// TIA Portal V17 export
// export: Created 2024-09-02T12:50:00.3255564Z, ExportSetting WithDefaults, DisplayName Totally Integrated Automation Portal, DisplayVersion V17, DisplayName TIA Portal Openness, DisplayVersion V17, DisplayName TIA Portal Version Control Interface, DisplayVersion V17, DisplayName STEP 7 Professional, DisplayVersion V17, DisplayName STEP 7 Safety, DisplayVersion V17, DisplayName WinCC Professional, DisplayVersion V17
FUNCTION_BLOCK "GraFB_Hand_31_40"   // FB1173, GRAPH
TITLE = GRAPH FB
AUTHOR : OlegFuehrus
FAMILY : SK
NAME : SK
VERSION : 0.1
// Hand functions / Handfunktionen
// stored: AcknowledgeErrorsRequired true, AutoNumber true, ExtensionBlockName LTLL_ManualGraphExt, GraphVersion 4.0, InitialValuesAcquisition false, IsIECCheckEnabled false, LanguageInNetworks LAD, LockOperatingMode false, PermanentILProcessingInMANMode true, SetENOAutomatically false, SkipSteps false, UDAEnableTagReadback false, WithAlarmHandling true
   // inherited from GRAPH_BASE
   VAR
      OFF_SQ_BASE : Bool;
   END_VAR
   VAR_INPUT
      OFF_SQ : Bool;
      INIT_SQ : Bool;
      ACK_EF : Bool;
      S_PREV : Bool;
      S_NEXT : Bool;
      SW_AUTO : Bool;
      SW_TAP : Bool;
      SW_MAN : Bool;
      S_SEL : Int;
      S_ON : Bool;
      S_OFF : Bool;
      T_PUSH : Bool;
   END_VAR
   VAR_OUTPUT
      S_NO : Int;
      S_MORE : Bool;
      S_ACTIVE : Bool;
      ERR_FLT : Bool;
      AUTO_ON : Bool;
      TAP_ON : Bool;
      MAN_ON : Bool;
   END_VAR
   VAR
      extBlock { S7_SetPoint := 'True'} : "LTLL_ManualGraphExt";
   END_VAR
   VAR_TEMP
      t_FrgHand : Bool;   // Freigabe Handbetrieb / Enable manual operation
      t_Service : Bool;   // Servicebetrieb aktiv / Service operation active
   END_VAR
BEGIN
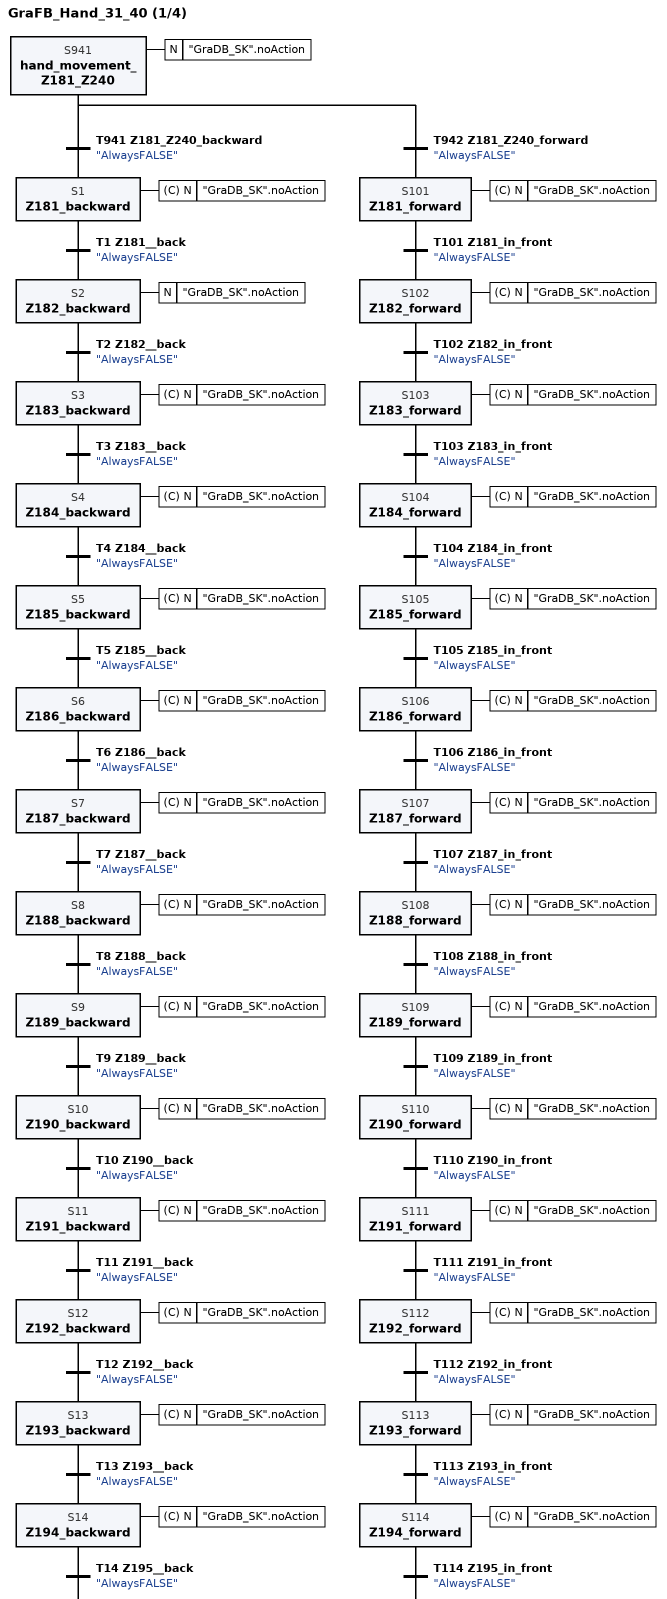
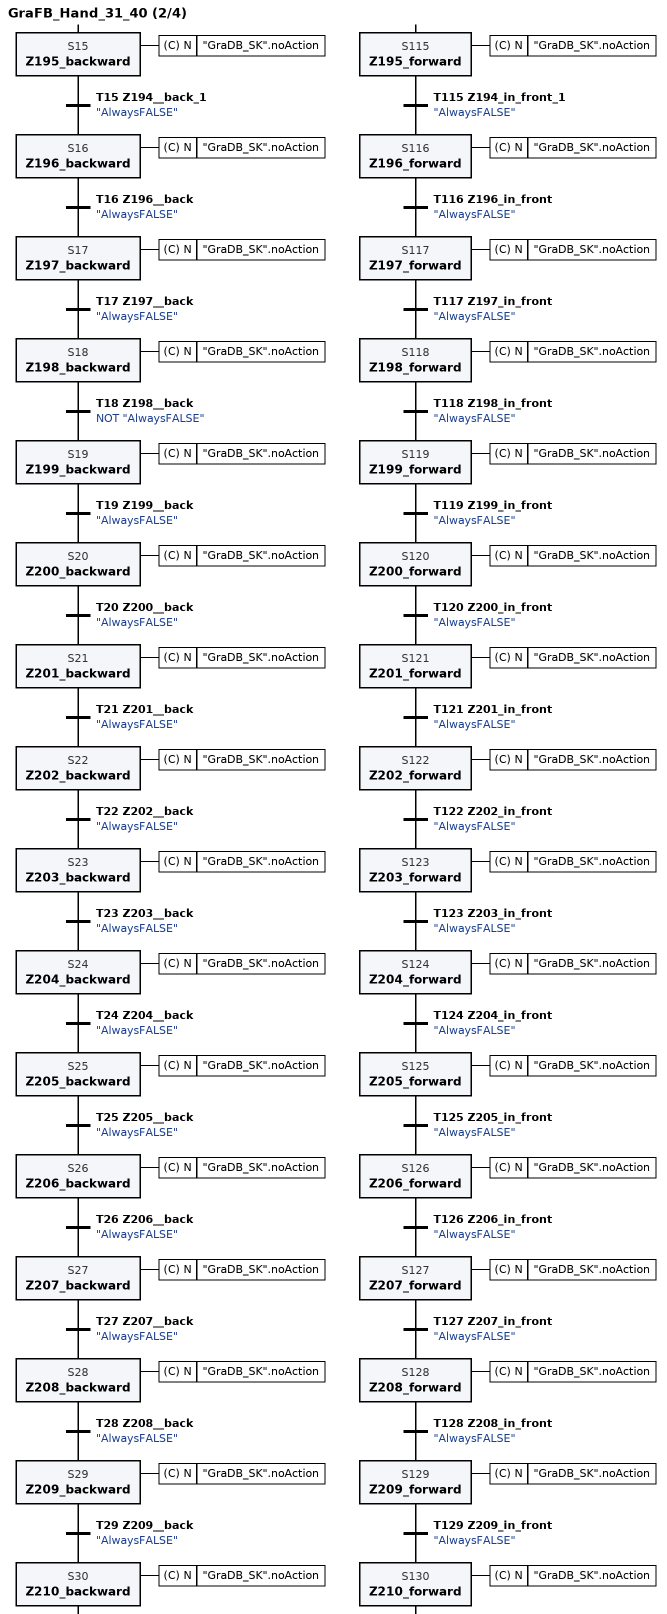
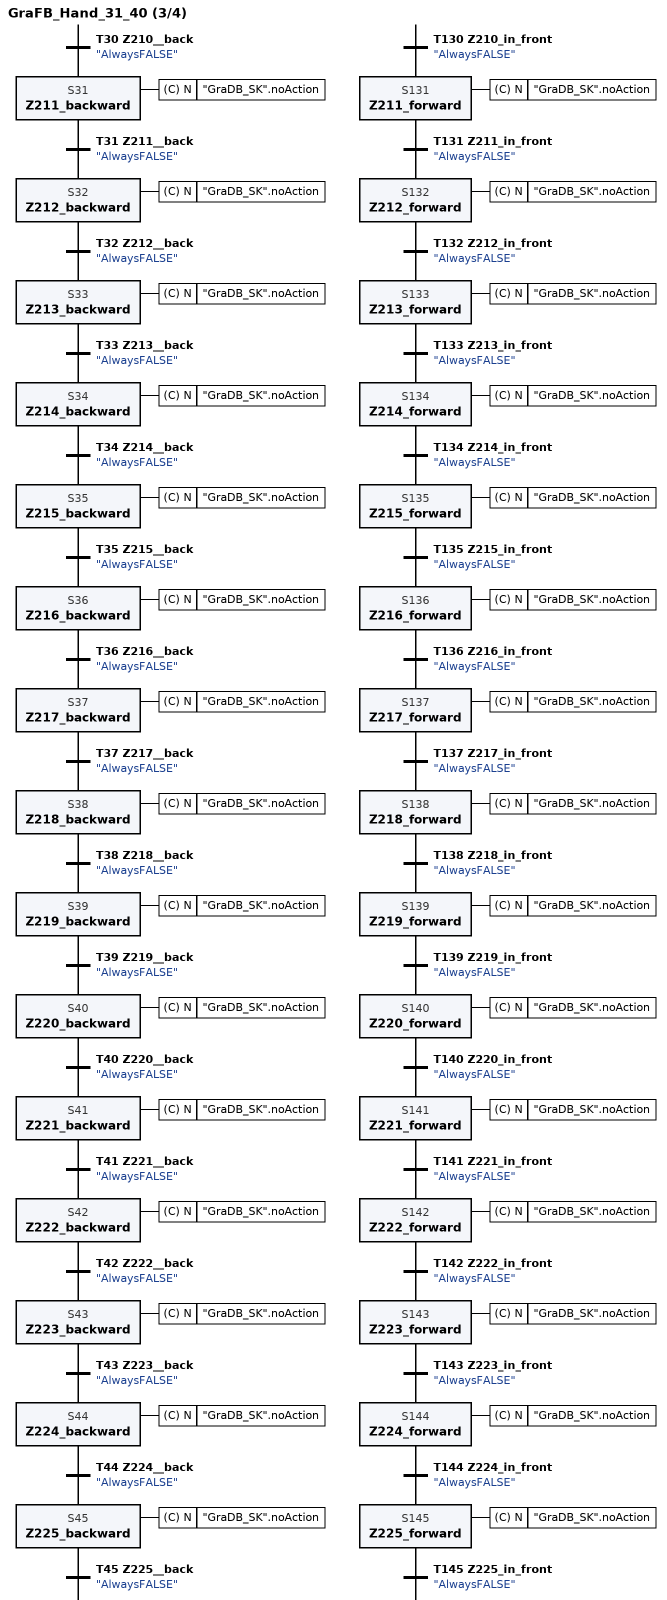
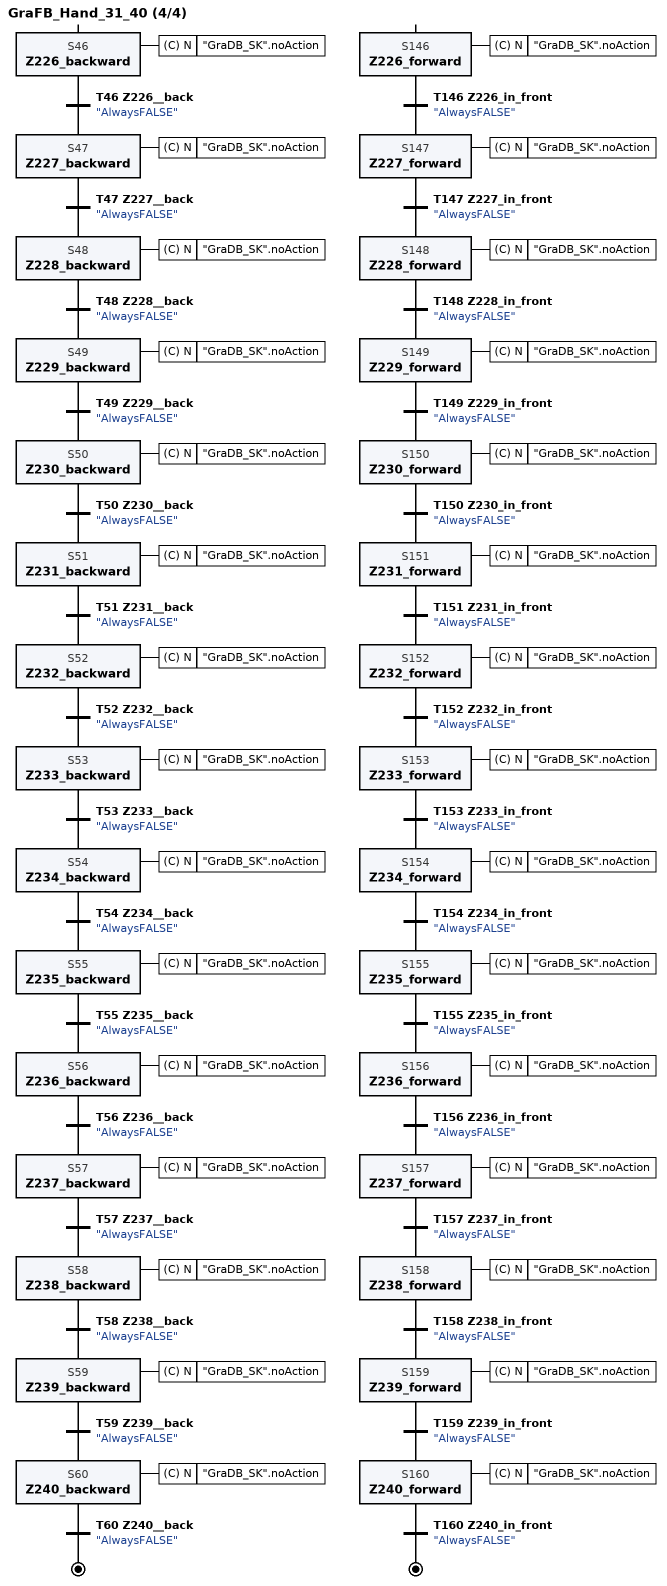
   // permanent pre-instructions
   NETWORK 1
   TITLE = HMI Lite Pass on data / HMI Lite Daten weiterreichen
      #extBlock.input := "LTLL_ManualGraphControl_OP70".screen[0].input;
   NETWORK 2
   TITLE = Instance DB Name query and pass on / Instanz DB Name abfragen und weiterreichen
      GetInstanceName(size := 0, OUT => #extBlock.input.instanceName);
   NETWORK 3
   TITLE = Interlocks Permanent machining, manual Approve and service / Interlocks Permanent Bearbeiten, Handfreigabe und Service
      IF NOT #RT_DATA.MOP.IL_PERM THEN #RT_DATA.MOP.IL_PERM := TRUE; END_IF;
      #t_FrgHand := "AnwDB_OperatingModes_OP70".BA[0]."mode_hand+start";
      #t_Service := "AnwDB_OperatingModes_OP70".BA[0].mode_service;

   // sequencer 1: Sequencer 1
   STEP hand_movement_Z181_Z240:   // S941, max time T#10S, warning time T#7S: Step commentary / Schrittkommentar
      interlock C := (none);   // hand_bereich_Z001_Z005
      supervision V := (none);   // hand_bereich_Z001_Z005
              N    "GraDB_SK".noAction
   END_STEP
   TRANSITION Z181_Z240_backward FROM hand_movement_Z181_Z240 TO Z181_backward   // T941
      := "AlwaysFALSE";
   END_TRANSITION
   TRANSITION Z181_Z240_forward FROM hand_movement_Z181_Z240 TO Z181_forward   // T942
      := "AlwaysFALSE";
   END_TRANSITION
   STEP Z181_backward:   // S1, max time T#10S, warning time T#7S
      interlock C := "AlwaysFALSE";   // Z181_zur
      supervision V := NOT #Z181__back.TT AND (#Z181_backward.T > T#5S);   // Z181_zur
      (C)     N    "GraDB_SK".noAction
   END_STEP
   TRANSITION Z181__back FROM Z181_backward TO Z182_backward   // T1
      := "AlwaysFALSE";
   END_TRANSITION
   STEP Z182_backward:   // S2, max time T#10S, warning time T#7S
      interlock C := "AlwaysFALSE";   // Z182_zur
      supervision V := NOT #Z182__back.TT AND (#Z182_backward.T > T#5S);   // Z182_zur
              N    "GraDB_SK".noAction
   END_STEP
   TRANSITION Z182__back FROM Z182_backward TO Z183_backward   // T2
      := "AlwaysFALSE";
   END_TRANSITION
   STEP Z183_backward:   // S3, max time T#10S, warning time T#7S
      interlock C := "AlwaysFALSE";   // Z183_zur
      supervision V := NOT #Z183__back.TT AND (#Z183_backward.T > T#5S);   // Z183_zur
      (C)     N    "GraDB_SK".noAction
   END_STEP
   TRANSITION Z183__back FROM Z183_backward TO Z184_backward   // T3
      := "AlwaysFALSE";
   END_TRANSITION
   STEP Z184_backward:   // S4, max time T#10S, warning time T#7S
      interlock C := "AlwaysFALSE";   // Z184_zur
      supervision V := NOT #Z184__back.TT AND (#Z184_backward.T > T#5S);   // Z184_zur
      (C)     N    "GraDB_SK".noAction
   END_STEP
   TRANSITION Z184__back FROM Z184_backward TO Z185_backward   // T4
      := "AlwaysFALSE";
   END_TRANSITION
   STEP Z185_backward:   // S5, max time T#10S, warning time T#7S
      interlock C := "AlwaysFALSE";   // Z185_zur
      supervision V := NOT #Z185__back.TT AND (#Z185_backward.T > T#5S);   // Z185_zur
      (C)     N    "GraDB_SK".noAction
   END_STEP
   TRANSITION Z185__back FROM Z185_backward TO Z186_backward   // T5
      := "AlwaysFALSE";
   END_TRANSITION
   STEP Z181_forward:   // S101, max time T#10S, warning time T#7S
      interlock C := "AlwaysFALSE";   // Z181_vor
      supervision V := NOT #Z181_in_front.TT AND (#Z181_forward.T > T#5S);   // Z181_vor
      (C)     N    "GraDB_SK".noAction
   END_STEP
   TRANSITION Z181_in_front FROM Z181_forward TO Z182_forward   // T101
      := "AlwaysFALSE";
   END_TRANSITION
   STEP Z182_forward:   // S102, max time T#10S, warning time T#7S
      interlock C := "AlwaysFALSE";   // Z182_vor
      supervision V := NOT #Z182_in_front.TT AND (#Z182_forward.T > T#5S);   // Z182_vor
      (C)     N    "GraDB_SK".noAction
   END_STEP
   TRANSITION Z182_in_front FROM Z182_forward TO Z183_forward   // T102
      := "AlwaysFALSE";
   END_TRANSITION
   STEP Z183_forward:   // S103, max time T#10S, warning time T#7S
      interlock C := "AlwaysFALSE";   // Z183_vor
      supervision V := NOT #Z183_in_front.TT AND (#Z183_forward.T > T#5S);   // Z183_vor
      (C)     N    "GraDB_SK".noAction
   END_STEP
   TRANSITION Z183_in_front FROM Z183_forward TO Z184_forward   // T103
      := "AlwaysFALSE";
   END_TRANSITION
   STEP Z184_forward:   // S104, max time T#10S, warning time T#7S
      interlock C := "AlwaysFALSE";   // Z184_vor
      supervision V := NOT #Z184_in_front.TT AND (#Z184_forward.T > T#5S);   // Z184_vor
      (C)     N    "GraDB_SK".noAction
   END_STEP
   TRANSITION Z184_in_front FROM Z184_forward TO Z185_forward   // T104
      := "AlwaysFALSE";
   END_TRANSITION
   STEP Z185_forward:   // S105, max time T#10S, warning time T#7S
      interlock C := "AlwaysFALSE";   // Z185_vor
      supervision V := NOT #Z185_in_front.TT AND (#Z185_forward.T > T#20S);   // Z185_vor
      (C)     N    "GraDB_SK".noAction
   END_STEP
   TRANSITION Z185_in_front FROM Z185_forward TO Z186_forward   // T105
      := "AlwaysFALSE";
   END_TRANSITION
   STEP Z186_backward:   // S6, max time T#10S, warning time T#7S: Cross transport 2 / Quertransport 2
      interlock C := "AlwaysFALSE";   // Z186_zur
      supervision V := NOT #Z186__back.TT AND (#Z186_backward.T > T#5S);   // Z186_zur
      (C)     N    "GraDB_SK".noAction
   END_STEP
   TRANSITION Z186__back FROM Z186_backward TO Z187_backward   // T6
      := "AlwaysFALSE";
   END_TRANSITION
   STEP Z187_backward:   // S7, max time T#10S, warning time T#7S
      interlock C := "AlwaysFALSE";   // Z187_zur
      supervision V := NOT #Z187__back.TT AND (#Z187_backward.T > T#5S);   // Z187_zur
      (C)     N    "GraDB_SK".noAction
   END_STEP
   TRANSITION Z187__back FROM Z187_backward TO Z188_backward   // T7
      := "AlwaysFALSE";
   END_TRANSITION
   STEP Z188_backward:   // S8, max time T#10S, warning time T#7S
      interlock C := "AlwaysFALSE";   // Z188_zur
      supervision V := NOT #Z188__back.TT AND (#Z188_backward.T > T#5S);   // Z188_zur
      (C)     N    "GraDB_SK".noAction
   END_STEP
   TRANSITION Z188__back FROM Z188_backward TO Z189_backward   // T8
      := "AlwaysFALSE";
   END_TRANSITION
   STEP Z189_backward:   // S9, max time T#10S, warning time T#7S
      interlock C := "AlwaysFALSE";   // Z189_zur
      supervision V := NOT #Z189__back.TT AND (#Z189_backward.T > T#5S);   // Z189_zur
      (C)     N    "GraDB_SK".noAction
   END_STEP
   TRANSITION Z189__back FROM Z189_backward TO Z190_backward   // T9
      := "AlwaysFALSE";
   END_TRANSITION
   STEP Z190_backward:   // S10, max time T#10S, warning time T#7S
      interlock C := "AlwaysFALSE";   // Z190_zur
      supervision V := NOT #Z190__back.TT AND (#Z190_backward.T > T#5S);   // Z190_zur
      (C)     N    "GraDB_SK".noAction
   END_STEP
   TRANSITION Z190__back FROM Z190_backward TO Z191_backward   // T10
      := "AlwaysFALSE";
   END_TRANSITION
   STEP Z186_forward:   // S106, max time T#10S, warning time T#7S
      interlock C := "AlwaysFALSE";   // Z186_vor
      supervision V := NOT #Z186_in_front.TT AND (#Z186_forward.T > T#5S);   // Z186_vor
      (C)     N    "GraDB_SK".noAction
   END_STEP
   TRANSITION Z186_in_front FROM Z186_forward TO Z187_forward   // T106
      := "AlwaysFALSE";
   END_TRANSITION
   STEP Z187_forward:   // S107, max time T#10S, warning time T#7S
      interlock C := "AlwaysFALSE";   // Z187_vor
      supervision V := NOT #Z187_in_front.TT AND (#Z187_forward.T > T#5S);   // Z187_vor
      (C)     N    "GraDB_SK".noAction
   END_STEP
   TRANSITION Z187_in_front FROM Z187_forward TO Z188_forward   // T107
      := "AlwaysFALSE";
   END_TRANSITION
   STEP Z188_forward:   // S108, max time T#10S, warning time T#7S
      interlock C := "AlwaysFALSE";   // Z188_vor
      supervision V := NOT #Z188_in_front.TT AND (#Z188_forward.T > T#5S);   // Z188_vor
      (C)     N    "GraDB_SK".noAction
   END_STEP
   TRANSITION Z188_in_front FROM Z188_forward TO Z189_forward   // T108
      := "AlwaysFALSE";
   END_TRANSITION
   STEP Z189_forward:   // S109, max time T#10S, warning time T#7S
      interlock C := "AlwaysFALSE";   // Z189_vor
      supervision V := NOT #Z189_in_front.TT AND (#Z189_forward.T > T#5S);   // Z189_vor
      (C)     N    "GraDB_SK".noAction
   END_STEP
   TRANSITION Z189_in_front FROM Z189_forward TO Z190_forward   // T109
      := "AlwaysFALSE";
   END_TRANSITION
   STEP Z190_forward:   // S110, max time T#10S, warning time T#7S
      interlock C := "AlwaysFALSE";   // Z190_vor
      supervision V := NOT #Z190_in_front.TT AND (#Z190_forward.T > T#5S);   // Z190_vor
      (C)     N    "GraDB_SK".noAction
   END_STEP
   TRANSITION Z190_in_front FROM Z190_forward TO Z191_forward   // T110
      := "AlwaysFALSE";
   END_TRANSITION
   STEP Z191_backward:   // S11, max time T#10S, warning time T#7S
      interlock C := "AlwaysFALSE";   // Z191_zur
      supervision V := NOT #Z191__back.TT AND (#Z191_backward.T > T#5S);   // Z191_zur
      (C)     N    "GraDB_SK".noAction
   END_STEP
   TRANSITION Z191__back FROM Z191_backward TO Z192_backward   // T11
      := "AlwaysFALSE";
   END_TRANSITION
   STEP Z192_backward:   // S12, max time T#10S, warning time T#7S
      interlock C := "AlwaysFALSE";   // Z192_zur
      supervision V := NOT #Z192__back.TT AND (#Z192_backward.T > T#5S);   // Z192_zur
      (C)     N    "GraDB_SK".noAction
   END_STEP
   TRANSITION Z192__back FROM Z192_backward TO Z193_backward   // T12
      := "AlwaysFALSE";
   END_TRANSITION
   STEP Z193_backward:   // S13, max time T#10S, warning time T#7S
      interlock C := "AlwaysFALSE";   // Z193_zur
      supervision V := NOT #Z193__back.TT AND (#Z193_backward.T > T#5S);   // Z193_zur
      (C)     N    "GraDB_SK".noAction
   END_STEP
   TRANSITION Z193__back FROM Z193_backward TO Z194_backward   // T13
      := "AlwaysFALSE";
   END_TRANSITION
   STEP Z194_backward:   // S14, max time T#10S, warning time T#7S
      interlock C := "AlwaysFALSE";   // Z194_zur
      supervision V := NOT #Z195__back.TT AND (#Z194_backward.T > T#5S);   // Z194_zur
      (C)     N    "GraDB_SK".noAction
   END_STEP
   TRANSITION Z195__back FROM Z194_backward TO Z195_backward   // T14
      := "AlwaysFALSE";
   END_TRANSITION
   STEP Z195_backward:   // S15, max time T#10S, warning time T#7S
      interlock C := "AlwaysFALSE";   // Z195_zur
      supervision V := NOT #Z196__back.TT AND (#Z195_backward.T > T#5S);   // Z195_zur
      (C)     N    "GraDB_SK".noAction
   END_STEP
   TRANSITION Z194__back_1 FROM Z195_backward TO Z196_backward   // T15
      := "AlwaysFALSE";
   END_TRANSITION
   STEP Z191_forward:   // S111, max time T#10S, warning time T#7S
      interlock C := "AlwaysFALSE";   // Z191_vor
      supervision V := NOT #Z191_in_front.TT AND (#Z191_forward.T > T#5S);   // Z191_vor
      (C)     N    "GraDB_SK".noAction
   END_STEP
   TRANSITION Z191_in_front FROM Z191_forward TO Z192_forward   // T111
      := "AlwaysFALSE";
   END_TRANSITION
   STEP Z192_forward:   // S112, max time T#10S, warning time T#7S
      interlock C := "AlwaysFALSE";   // Z192_vor
      supervision V := NOT #Z192_in_front.TT AND (#Z192_forward.T > T#5S);   // Z192_vor
      (C)     N    "GraDB_SK".noAction
   END_STEP
   TRANSITION Z192_in_front FROM Z192_forward TO Z193_forward   // T112
      := "AlwaysFALSE";
   END_TRANSITION
   STEP Z193_forward:   // S113, max time T#10S, warning time T#7S
      interlock C := "AlwaysFALSE";   // Z193_vor
      supervision V := NOT #Z193_in_front.TT AND (#Z193_forward.T > T#5S);   // Z193_vor
      (C)     N    "GraDB_SK".noAction
   END_STEP
   TRANSITION Z193_in_front FROM Z193_forward TO Z194_forward   // T113
      := "AlwaysFALSE";
   END_TRANSITION
   STEP Z194_forward:   // S114, max time T#10S, warning time T#7S
      interlock C := "AlwaysFALSE";   // Z194_vor
      supervision V := NOT #Z195_in_front.TT AND (#Z194_forward.T > T#5S);   // Z194_vor
      (C)     N    "GraDB_SK".noAction
   END_STEP
   TRANSITION Z195_in_front FROM Z194_forward TO Z195_forward   // T114
      := "AlwaysFALSE";
   END_TRANSITION
   STEP Z195_forward:   // S115, max time T#10S, warning time T#7S
      interlock C := "AlwaysFALSE";   // Z195_vor
      supervision V := NOT #Z196_in_front.TT AND (#Z195_forward.T > T#5S);   // Z195_vor
      (C)     N    "GraDB_SK".noAction
   END_STEP
   TRANSITION Z194_in_front_1 FROM Z195_forward TO Z196_forward   // T115
      := "AlwaysFALSE";
   END_TRANSITION
   STEP Z196_backward:   // S16, max time T#10S, warning time T#7S
      interlock C := "AlwaysFALSE";   // Z196_zur
      supervision V := NOT #Z196__back.TT AND (#Z196_backward.T > T#5S);   // Z196_zur
      (C)     N    "GraDB_SK".noAction
   END_STEP
   TRANSITION Z196__back FROM Z196_backward TO Z197_backward   // T16
      := "AlwaysFALSE";
   END_TRANSITION
   STEP Z197_backward:   // S17, max time T#10S, warning time T#7S
      interlock C := "AlwaysFALSE";   // Z197_zur
      supervision V := NOT #Z197__back.TT AND (#Z197_backward.T > T#5S);   // Z197_zur
      (C)     N    "GraDB_SK".noAction
   END_STEP
   TRANSITION Z197__back FROM Z197_backward TO Z198_backward   // T17
      := "AlwaysFALSE";
   END_TRANSITION
   STEP Z198_backward:   // S18, max time T#10S, warning time T#7S
      interlock C := "AlwaysFALSE";   // Z198_zur
      supervision V := NOT #Z198__back.TT AND (#Z198_backward.T > T#5S);   // Z198_zur
      (C)     N    "GraDB_SK".noAction
   END_STEP
   TRANSITION Z198__back FROM Z198_backward TO Z199_backward   // T18
      := NOT "AlwaysFALSE";
   END_TRANSITION
   STEP Z199_backward:   // S19, max time T#10S, warning time T#7S
      interlock C := "AlwaysFALSE";   // Z199_zur
      supervision V := NOT #Z199__back.TT AND (#Z199_backward.T > T#5S);   // Z199_zur
      (C)     N    "GraDB_SK".noAction
   END_STEP
   TRANSITION Z199__back FROM Z199_backward TO Z200_backward   // T19
      := "AlwaysFALSE";
   END_TRANSITION
   STEP Z200_backward:   // S20, max time T#10S, warning time T#7S
      interlock C := "AlwaysFALSE";   // Z200_zur
      supervision V := NOT #Z200__back.TT AND (#Z200_backward.T > T#5S);   // Z2000_zur
      (C)     N    "GraDB_SK".noAction
   END_STEP
   TRANSITION Z200__back FROM Z200_backward TO Z201_backward   // T20
      := "AlwaysFALSE";
   END_TRANSITION
   STEP Z196_forward:   // S116, max time T#10S, warning time T#7S
      interlock C := "AlwaysFALSE";   // Z196_vor
      supervision V := NOT #Z196_in_front.TT AND (#Z196_forward.T > T#5S);   // Z196_vor
      (C)     N    "GraDB_SK".noAction
   END_STEP
   TRANSITION Z196_in_front FROM Z196_forward TO Z197_forward   // T116
      := "AlwaysFALSE";
   END_TRANSITION
   STEP Z197_forward:   // S117, max time T#10S, warning time T#7S
      interlock C := "AlwaysFALSE";   // Z197_vor
      supervision V := NOT #Z197_in_front.TT AND (#Z197_forward.T > T#5S);   // Z197_vor
      (C)     N    "GraDB_SK".noAction
   END_STEP
   TRANSITION Z197_in_front FROM Z197_forward TO Z198_forward   // T117
      := "AlwaysFALSE";
   END_TRANSITION
   STEP Z198_forward:   // S118, max time T#10S, warning time T#7S
      interlock C := "AlwaysFALSE";   // Z198_vor
      supervision V := NOT #Z198_in_front.TT AND (#Z198_forward.T > T#5S);   // Z198_vor
      (C)     N    "GraDB_SK".noAction
   END_STEP
   TRANSITION Z198_in_front FROM Z198_forward TO Z199_forward   // T118
      := "AlwaysFALSE";
   END_TRANSITION
   STEP Z199_forward:   // S119, max time T#10S, warning time T#7S
      interlock C := "AlwaysFALSE";   // Z199_vor
      supervision V := NOT #Z199_in_front.TT AND (#Z199_forward.T > T#5S);   // Z199_vor
      (C)     N    "GraDB_SK".noAction
   END_STEP
   TRANSITION Z199_in_front FROM Z199_forward TO Z200_forward   // T119
      := "AlwaysFALSE";
   END_TRANSITION
   STEP Z200_forward:   // S120, max time T#10S, warning time T#7S
      interlock C := "AlwaysFALSE";   // Z200_vor
      supervision V := NOT #Z200_in_front.TT AND (#Z200_forward.T > T#5S);   // Z200_vor
      (C)     N    "GraDB_SK".noAction
   END_STEP
   TRANSITION Z200_in_front FROM Z200_forward TO Z201_forward   // T120
      := "AlwaysFALSE";
   END_TRANSITION
   STEP Z201_backward:   // S21, max time T#10S, warning time T#7S
      interlock C := "AlwaysFALSE";   // Z201_zur
      supervision V := NOT #Z201__back.TT AND (#Z201_backward.T > T#10S);   // Z201_zur
      (C)     N    "GraDB_SK".noAction
   END_STEP
   TRANSITION Z201__back FROM Z201_backward TO Z202_backward   // T21
      := "AlwaysFALSE";
   END_TRANSITION
   STEP Z202_backward:   // S22, max time T#10S, warning time T#7S
      interlock C := "AlwaysFALSE";   // Z202_zur
      supervision V := NOT #Z202__back.TT AND (#Z202_backward.T > T#10S);   // Z202_zur
      (C)     N    "GraDB_SK".noAction
   END_STEP
   TRANSITION Z202__back FROM Z202_backward TO Z203_backward   // T22
      := "AlwaysFALSE";
   END_TRANSITION
   STEP Z203_backward:   // S23, max time T#10S, warning time T#7S
      interlock C := "AlwaysFALSE";   // Z203_zur
      supervision V := NOT #Z203__back.TT AND (#Z203_backward.T > T#10S);   // Z203_zur
      (C)     N    "GraDB_SK".noAction
   END_STEP
   TRANSITION Z203__back FROM Z203_backward TO Z204_backward   // T23
      := "AlwaysFALSE";
   END_TRANSITION
   STEP Z204_backward:   // S24, max time T#10S, warning time T#7S
      interlock C := "AlwaysFALSE";   // Z204_zur
      supervision V := NOT #Z204__back.TT AND (#Z204_backward.T > T#5S);   // Z204_zur
      (C)     N    "GraDB_SK".noAction
   END_STEP
   TRANSITION Z204__back FROM Z204_backward TO Z205_backward   // T24
      := "AlwaysFALSE";
   END_TRANSITION
   STEP Z205_backward:   // S25, max time T#10S, warning time T#7S
      interlock C := "AlwaysFALSE";   // Z205_zur
      supervision V := NOT #Z205__back.TT AND (#Z205_backward.T > T#5S);   // Z205_zur
      (C)     N    "GraDB_SK".noAction
   END_STEP
   TRANSITION Z205__back FROM Z205_backward TO Z206_backward   // T25
      := "AlwaysFALSE";
   END_TRANSITION
   STEP Z201_forward:   // S121, max time T#10S, warning time T#7S
      interlock C := "AlwaysFALSE";   // Z201_vor
      supervision V := NOT #Z201_in_front.TT AND (#Z201_forward.T > T#5S);   // Z201_vor
      (C)     N    "GraDB_SK".noAction
   END_STEP
   TRANSITION Z201_in_front FROM Z201_forward TO Z202_forward   // T121
      := "AlwaysFALSE";
   END_TRANSITION
   STEP Z202_forward:   // S122, max time T#10S, warning time T#7S
      interlock C := "AlwaysFALSE";   // Z202_vor
      supervision V := NOT #Z202_in_front.TT AND (#Z202_forward.T > T#10S);   // Z202_vor
      (C)     N    "GraDB_SK".noAction
   END_STEP
   TRANSITION Z202_in_front FROM Z202_forward TO Z203_forward   // T122
      := "AlwaysFALSE";
   END_TRANSITION
   STEP Z203_forward:   // S123, max time T#10S, warning time T#7S
      interlock C := "AlwaysFALSE";   // Z203_vor
      supervision V := NOT #Z203_in_front.TT AND (#Z203_forward.T > T#10S);   // Z203_vor
      (C)     N    "GraDB_SK".noAction
   END_STEP
   TRANSITION Z203_in_front FROM Z203_forward TO Z204_forward   // T123
      := "AlwaysFALSE";
   END_TRANSITION
   STEP Z204_forward:   // S124, max time T#10S, warning time T#7S
      interlock C := "AlwaysFALSE";   // Z204_vor
      supervision V := NOT #Z204_in_front.TT AND (#Z204_forward.T > T#5S);   // Z204_vor
      (C)     N    "GraDB_SK".noAction
   END_STEP
   TRANSITION Z204_in_front FROM Z204_forward TO Z205_forward   // T124
      := "AlwaysFALSE";
   END_TRANSITION
   STEP Z205_forward:   // S125, max time T#10S, warning time T#7S
      interlock C := "AlwaysFALSE";   // Z205_vor
      supervision V := NOT #Z205_in_front.TT AND (#Z205_forward.T > T#5S);   // Z205_vor
      (C)     N    "GraDB_SK".noAction
   END_STEP
   TRANSITION Z205_in_front FROM Z205_forward TO Z206_forward   // T125
      := "AlwaysFALSE";
   END_TRANSITION
   STEP Z206_backward:   // S26, max time T#10S, warning time T#7S
      interlock C := "AlwaysFALSE";   // Z206_zur
      supervision V := NOT #Z206__back.TT AND (#Z206_backward.T > T#5S);   // Z206_zur
      (C)     N    "GraDB_SK".noAction
   END_STEP
   TRANSITION Z206__back FROM Z206_backward TO Z207_backward   // T26
      := "AlwaysFALSE";
   END_TRANSITION
   STEP Z207_backward:   // S27, max time T#10S, warning time T#7S
      interlock C := "AlwaysFALSE";   // Z207_zur
      supervision V := NOT #Z207__back.TT AND (#Z207_backward.T > T#5S);   // Z207_zur
      (C)     N    "GraDB_SK".noAction
   END_STEP
   TRANSITION Z207__back FROM Z207_backward TO Z208_backward   // T27
      := "AlwaysFALSE";
   END_TRANSITION
   STEP Z208_backward:   // S28, max time T#10S, warning time T#7S
      interlock C := "AlwaysFALSE";   // Z208_zur
      supervision V := NOT #Z208__back.TT AND (#Z208_backward.T > T#5S);   // Z208_zur
      (C)     N    "GraDB_SK".noAction
   END_STEP
   TRANSITION Z208__back FROM Z208_backward TO Z209_backward   // T28
      := "AlwaysFALSE";
   END_TRANSITION
   STEP Z209_backward:   // S29, max time T#10S, warning time T#7S
      interlock C := "AlwaysFALSE";   // Z209_zur
      supervision V := NOT #Z209__back.TT AND (#Z209_backward.T > T#5S);   // Z209_zur
      (C)     N    "GraDB_SK".noAction
   END_STEP
   TRANSITION Z209__back FROM Z209_backward TO Z210_backward   // T29
      := "AlwaysFALSE";
   END_TRANSITION
   STEP Z210_backward:   // S30, max time T#10S, warning time T#7S
      interlock C := "AlwaysFALSE";   // Z210_zur
      supervision V := NOT #Z210__back.TT AND (#Z210_backward.T > T#5S);   // Z210_zur
      (C)     N    "GraDB_SK".noAction
   END_STEP
   TRANSITION Z210__back FROM Z210_backward TO Z211_backward   // T30
      := "AlwaysFALSE";
   END_TRANSITION
   STEP Z206_forward:   // S126, max time T#10S, warning time T#7S
      interlock C := "AlwaysFALSE";   // Z206_vor
      supervision V := NOT #Z206_in_front.TT AND (#Z206_forward.T > T#5S);   // Z206_vor
      (C)     N    "GraDB_SK".noAction
   END_STEP
   TRANSITION Z206_in_front FROM Z206_forward TO Z207_forward   // T126
      := "AlwaysFALSE";
   END_TRANSITION
   STEP Z207_forward:   // S127, max time T#10S, warning time T#7S
      interlock C := "AlwaysFALSE";   // Z207_vor
      supervision V := NOT #Z207_in_front.TT AND (#Z207_forward.T > T#5S);   // Z207_vor
      (C)     N    "GraDB_SK".noAction
   END_STEP
   TRANSITION Z207_in_front FROM Z207_forward TO Z208_forward   // T127
      := "AlwaysFALSE";
   END_TRANSITION
   STEP Z208_forward:   // S128, max time T#10S, warning time T#7S
      interlock C := "AlwaysFALSE";   // Z208_vor
      supervision V := NOT #Z208_in_front.TT AND (#Z208_forward.T > T#5S);   // Z208_vor
      (C)     N    "GraDB_SK".noAction
   END_STEP
   TRANSITION Z208_in_front FROM Z208_forward TO Z209_forward   // T128
      := "AlwaysFALSE";
   END_TRANSITION
   STEP Z209_forward:   // S129, max time T#10S, warning time T#7S
      interlock C := "AlwaysFALSE";   // Z209_vor
      supervision V := NOT #Z209_in_front.TT AND (#Z209_forward.T > T#5S);   // Z209_vor
      (C)     N    "GraDB_SK".noAction
   END_STEP
   TRANSITION Z209_in_front FROM Z209_forward TO Z210_forward   // T129
      := "AlwaysFALSE";
   END_TRANSITION
   STEP Z210_forward:   // S130, max time T#10S, warning time T#7S
      interlock C := "AlwaysFALSE";   // Z210_vor
      supervision V := NOT #Z210_in_front.TT AND (#Z210_forward.T > T#5S);   // Z210_vor
      (C)     N    "GraDB_SK".noAction
   END_STEP
   TRANSITION Z210_in_front FROM Z210_forward TO Z211_forward   // T130
      := "AlwaysFALSE";
   END_TRANSITION
   STEP Z211_backward:   // S31, max time T#10S, warning time T#7S: Step commentary / Schrittkommentar
      interlock C := "AlwaysFALSE";   // Z211_zur
      supervision V := NOT #Z211__back.TT AND (#Z211_backward.T > T#5S);   // Z211_zur
      (C)     N    "GraDB_SK".noAction
   END_STEP
   TRANSITION Z211__back FROM Z211_backward TO Z212_backward   // T31
      := "AlwaysFALSE";
   END_TRANSITION
   STEP Z212_backward:   // S32, max time T#10S, warning time T#7S: Step commentary / Schrittkommentar
      interlock C := "AlwaysFALSE";   // Z212_zur
      supervision V := NOT #Z212__back.TT AND (#Z212_backward.T > T#5S);   // Z212_zur
      (C)     N    "GraDB_SK".noAction
   END_STEP
   TRANSITION Z212__back FROM Z212_backward TO Z213_backward   // T32
      := "AlwaysFALSE";
   END_TRANSITION
   STEP Z213_backward:   // S33, max time T#10S, warning time T#7S: Step commentary / Schrittkommentar
      interlock C := "AlwaysFALSE";   // Z213_zur
      supervision V := NOT #Z213__back.TT AND (#Z213_backward.T > T#5S);   // Z213_zur
      (C)     N    "GraDB_SK".noAction
   END_STEP
   TRANSITION Z213__back FROM Z213_backward TO Z214_backward   // T33
      := "AlwaysFALSE";
   END_TRANSITION
   STEP Z214_backward:   // S34, max time T#10S, warning time T#7S: Step commentary / Schrittkommentar
      interlock C := "AlwaysFALSE";   // Z034_zur
      supervision V := NOT #Z214__back.TT AND (#Z214_backward.T > T#5S);   // Z034_zur
      (C)     N    "GraDB_SK".noAction
   END_STEP
   TRANSITION Z214__back FROM Z214_backward TO Z215_backward   // T34
      := "AlwaysFALSE";
   END_TRANSITION
   STEP Z215_backward:   // S35, max time T#10S, warning time T#7S: Step commentary / Schrittkommentar
      interlock C := "AlwaysFALSE";   // Z215_zur
      supervision V := NOT #Z215__back.TT AND (#Z215_backward.T > T#5S);   // Z215_zur
      (C)     N    "GraDB_SK".noAction
   END_STEP
   TRANSITION Z215__back FROM Z215_backward TO Z216_backward   // T35
      := "AlwaysFALSE";
   END_TRANSITION
   STEP Z211_forward:   // S131, max time T#10S, warning time T#7S: Step commentary / Schrittkommentar
      interlock C := "AlwaysFALSE";   // Z211_vor
      supervision V := NOT #Z211_in_front.TT AND (#Z211_forward.T > T#5S);   // Z211_vor
      (C)     N    "GraDB_SK".noAction
   END_STEP
   TRANSITION Z211_in_front FROM Z211_forward TO Z212_forward   // T131
      := "AlwaysFALSE";
   END_TRANSITION
   STEP Z212_forward:   // S132, max time T#10S, warning time T#7S: Step commentary / Schrittkommentar
      interlock C := "AlwaysFALSE";   // Z212_vor
      supervision V := NOT #Z212_in_front.TT AND (#Z212_forward.T > T#5S);   // Z212_vor
      (C)     N    "GraDB_SK".noAction
   END_STEP
   TRANSITION Z212_in_front FROM Z212_forward TO Z213_forward   // T132
      := "AlwaysFALSE";
   END_TRANSITION
   STEP Z213_forward:   // S133, max time T#10S, warning time T#7S: Step commentary / Schrittkommentar
      interlock C := "AlwaysFALSE";   // Z213_vor
      supervision V := NOT #Z213_in_front.TT AND (#Z213_forward.T > T#5S);   // Z213_vor
      (C)     N    "GraDB_SK".noAction
   END_STEP
   TRANSITION Z213_in_front FROM Z213_forward TO Z214_forward   // T133
      := "AlwaysFALSE";
   END_TRANSITION
   STEP Z214_forward:   // S134, max time T#10S, warning time T#7S: Step commentary / Schrittkommentar
      interlock C := "AlwaysFALSE";   // Z034_vor
      supervision V := NOT #Z214_in_front.TT AND (#Z214_forward.T > T#5S);   // Z034_vor
      (C)     N    "GraDB_SK".noAction
   END_STEP
   TRANSITION Z214_in_front FROM Z214_forward TO Z215_forward   // T134
      := "AlwaysFALSE";
   END_TRANSITION
   STEP Z215_forward:   // S135, max time T#10S, warning time T#7S: Step commentary / Schrittkommentar
      interlock C := "AlwaysFALSE";   // Z215_vor
      supervision V := NOT #Z215_in_front.TT AND (#Z215_forward.T > T#5S);   // Z215_vor
      (C)     N    "GraDB_SK".noAction
   END_STEP
   TRANSITION Z215_in_front FROM Z215_forward TO Z216_forward   // T135
      := "AlwaysFALSE";
   END_TRANSITION
   STEP Z216_backward:   // S36, max time T#10S, warning time T#7S: Step commentary / Schrittkommentar
      interlock C := "AlwaysFALSE";   // Z216_zur
      supervision V := NOT #Z216__back.TT AND (#Z216_backward.T > T#5S);   // Z216_zur
      (C)     N    "GraDB_SK".noAction
   END_STEP
   TRANSITION Z216__back FROM Z216_backward TO Z217_backward   // T36
      := "AlwaysFALSE";
   END_TRANSITION
   STEP Z217_backward:   // S37, max time T#10S, warning time T#7S: Step commentary / Schrittkommentar
      interlock C := "AlwaysFALSE";   // Z217_zur
      supervision V := NOT #Z217__back.TT AND (#Z217_backward.T > T#5S);   // Z217_zur
      (C)     N    "GraDB_SK".noAction
   END_STEP
   TRANSITION Z217__back FROM Z217_backward TO Z218_backward   // T37
      := "AlwaysFALSE";
   END_TRANSITION
   STEP Z218_backward:   // S38, max time T#10S, warning time T#7S: Step commentary / Schrittkommentar
      interlock C := "AlwaysFALSE";   // Z218_zur
      supervision V := NOT #Z218__back.TT AND (#Z218_backward.T > T#5S);   // Z218_zur
      (C)     N    "GraDB_SK".noAction
   END_STEP
   TRANSITION Z218__back FROM Z218_backward TO Z219_backward   // T38
      := "AlwaysFALSE";
   END_TRANSITION
   STEP Z219_backward:   // S39, max time T#10S, warning time T#7S: Step commentary / Schrittkommentar
      interlock C := "AlwaysFALSE";   // Z219_zur
      supervision V := NOT #Z219__back.TT AND (#Z219_backward.T > T#5S);   // Z219_zur
      (C)     N    "GraDB_SK".noAction
   END_STEP
   TRANSITION Z219__back FROM Z219_backward TO Z220_backward   // T39
      := "AlwaysFALSE";
   END_TRANSITION
   STEP Z220_backward:   // S40, max time T#10S, warning time T#7S: Step commentary / Schrittkommentar
      interlock C := "AlwaysFALSE";   // Z220_zur
      supervision V := NOT #Z220__back.TT AND (#Z220_backward.T > T#5S);   // Z220_zur
      (C)     N    "GraDB_SK".noAction
   END_STEP
   TRANSITION Z220__back FROM Z220_backward TO Z221_backward   // T40
      := "AlwaysFALSE";
   END_TRANSITION
   STEP Z216_forward:   // S136, max time T#10S, warning time T#7S: Step commentary / Schrittkommentar
      interlock C := "AlwaysFALSE";   // Z216_vor
      supervision V := NOT #Z216_in_front.TT AND (#Z216_forward.T > T#5S);   // Z216_vor
      (C)     N    "GraDB_SK".noAction
   END_STEP
   TRANSITION Z216_in_front FROM Z216_forward TO Z217_forward   // T136
      := "AlwaysFALSE";
   END_TRANSITION
   STEP Z217_forward:   // S137, max time T#10S, warning time T#7S: Step commentary / Schrittkommentar
      interlock C := "AlwaysFALSE";   // Z217_vor
      supervision V := NOT #Z217_in_front.TT AND (#Z217_forward.T > T#5S);   // Z217_vor
      (C)     N    "GraDB_SK".noAction
   END_STEP
   TRANSITION Z217_in_front FROM Z217_forward TO Z218_forward   // T137
      := "AlwaysFALSE";
   END_TRANSITION
   STEP Z218_forward:   // S138, max time T#10S, warning time T#7S: Step commentary / Schrittkommentar
      interlock C := "AlwaysFALSE";   // Z218_vor
      supervision V := NOT #Z218_in_front.TT AND (#Z218_forward.T > T#5S);   // Z218_vor
      (C)     N    "GraDB_SK".noAction
   END_STEP
   TRANSITION Z218_in_front FROM Z218_forward TO Z219_forward   // T138
      := "AlwaysFALSE";
   END_TRANSITION
   STEP Z219_forward:   // S139, max time T#10S, warning time T#7S: Step commentary / Schrittkommentar
      interlock C := "AlwaysFALSE";   // Z219_vor
      supervision V := NOT #Z219_in_front.TT AND (#Z219_forward.T > T#5S);   // Z219_vor
      (C)     N    "GraDB_SK".noAction
   END_STEP
   TRANSITION Z219_in_front FROM Z219_forward TO Z220_forward   // T139
      := "AlwaysFALSE";
   END_TRANSITION
   STEP Z220_forward:   // S140, max time T#10S, warning time T#7S: Step commentary / Schrittkommentar
      interlock C := "AlwaysFALSE";   // Z220_vor
      supervision V := NOT #Z220_in_front.TT AND (#Z220_forward.T > T#5S);   // Z220_vor
      (C)     N    "GraDB_SK".noAction
   END_STEP
   TRANSITION Z220_in_front FROM Z220_forward TO Z221_forward   // T140
      := "AlwaysFALSE";
   END_TRANSITION
   STEP Z221_backward:   // S41, max time T#10S, warning time T#7S: Step commentary / Schrittkommentar
      interlock C := "AlwaysFALSE";   // Z221_zur
      supervision V := NOT #Z221__back.TT AND (#Z221_backward.T > T#5S);   // Z221_zur
      (C)     N    "GraDB_SK".noAction
   END_STEP
   TRANSITION Z221__back FROM Z221_backward TO Z222_backward   // T41
      := "AlwaysFALSE";
   END_TRANSITION
   STEP Z222_backward:   // S42, max time T#10S, warning time T#7S: Step commentary / Schrittkommentar
      interlock C := "AlwaysFALSE";   // Z222_zur
      supervision V := NOT #Z222__back.TT AND (#Z222_backward.T > T#5S);   // Z222_zur
      (C)     N    "GraDB_SK".noAction
   END_STEP
   TRANSITION Z222__back FROM Z222_backward TO Z223_backward   // T42
      := "AlwaysFALSE";
   END_TRANSITION
   STEP Z223_backward:   // S43, max time T#10S, warning time T#7S: Step commentary / Schrittkommentar
      interlock C := "AlwaysFALSE";   // Z223_zur
      supervision V := NOT #Z223__back.TT AND (#Z223_backward.T > T#5S);   // Z223_zur
      (C)     N    "GraDB_SK".noAction
   END_STEP
   TRANSITION Z223__back FROM Z223_backward TO Z224_backward   // T43
      := "AlwaysFALSE";
   END_TRANSITION
   STEP Z224_backward:   // S44, max time T#10S, warning time T#7S: Step commentary / Schrittkommentar
      interlock C := "AlwaysFALSE";   // Z224_zur
      supervision V := NOT #Z224__back.TT AND (#Z224_backward.T > T#5S);   // Z224_zur
      (C)     N    "GraDB_SK".noAction
   END_STEP
   TRANSITION Z224__back FROM Z224_backward TO Z225_backward   // T44
      := "AlwaysFALSE";
   END_TRANSITION
   STEP Z225_backward:   // S45, max time T#10S, warning time T#7S: Step commentary / Schrittkommentar
      interlock C := "AlwaysFALSE";   // Z225_zur
      supervision V := NOT #Z225__back.TT AND (#Z225_backward.T > T#5S);   // Z225_zur
      (C)     N    "GraDB_SK".noAction
   END_STEP
   TRANSITION Z225__back FROM Z225_backward TO Z226_backward   // T45
      := "AlwaysFALSE";
   END_TRANSITION
   STEP Z221_forward:   // S141, max time T#10S, warning time T#7S
      interlock C := "AlwaysFALSE";   // Z221_vor
      supervision V := NOT #Z221_in_front.TT AND (#Z221_forward.T > T#5S);   // Z221_vor
      (C)     N    "GraDB_SK".noAction
   END_STEP
   TRANSITION Z221_in_front FROM Z221_forward TO Z222_forward   // T141
      := "AlwaysFALSE";
   END_TRANSITION
   STEP Z222_forward:   // S142, max time T#10S, warning time T#7S
      interlock C := "AlwaysFALSE";   // Z222_vor
      supervision V := NOT #Z222_in_front.TT AND (#Z222_forward.T > T#5S);   // Z222_vor
      (C)     N    "GraDB_SK".noAction
   END_STEP
   TRANSITION Z222_in_front FROM Z222_forward TO Z223_forward   // T142
      := "AlwaysFALSE";
   END_TRANSITION
   STEP Z223_forward:   // S143, max time T#10S, warning time T#7S
      interlock C := "AlwaysFALSE";   // Z223_vor
      supervision V := NOT #Z223_in_front.TT AND (#Z223_forward.T > T#5S);   // Z223_vor
      (C)     N    "GraDB_SK".noAction
   END_STEP
   TRANSITION Z223_in_front FROM Z223_forward TO Z224_forward   // T143
      := "AlwaysFALSE";
   END_TRANSITION
   STEP Z224_forward:   // S144, max time T#10S, warning time T#7S
      interlock C := "AlwaysFALSE";   // Z224_vor
      supervision V := NOT #Z224_in_front.TT AND (#Z224_forward.T > T#5S);   // Z224_vor
      (C)     N    "GraDB_SK".noAction
   END_STEP
   TRANSITION Z224_in_front FROM Z224_forward TO Z225_forward   // T144
      := "AlwaysFALSE";
   END_TRANSITION
   STEP Z225_forward:   // S145, max time T#10S, warning time T#7S
      interlock C := "AlwaysFALSE";   // Z225_vor
      supervision V := NOT #Z225_in_front.TT AND (#Z225_forward.T > T#5S);   // Z225_vor
      (C)     N    "GraDB_SK".noAction
   END_STEP
   TRANSITION Z225_in_front FROM Z225_forward TO Z226_forward   // T145
      := "AlwaysFALSE";
   END_TRANSITION
   STEP Z226_backward:   // S46, max time T#10S, warning time T#7S: Step commentary / Schrittkommentar
      interlock C := "AlwaysFALSE";   // Z226_zur
      supervision V := NOT #Z226__back.TT AND (#Z226_backward.T > T#5S);   // Z226_zur
      (C)     N    "GraDB_SK".noAction
   END_STEP
   TRANSITION Z226__back FROM Z226_backward TO Z227_backward   // T46
      := "AlwaysFALSE";
   END_TRANSITION
   STEP Z227_backward:   // S47, max time T#10S, warning time T#7S: Step commentary / Schrittkommentar
      interlock C := "AlwaysFALSE";   // Z227_zur
      supervision V := NOT #Z227__back.TT AND (#Z227_backward.T > T#5S);   // Z227_zur
      (C)     N    "GraDB_SK".noAction
   END_STEP
   TRANSITION Z227__back FROM Z227_backward TO Z228_backward   // T47
      := "AlwaysFALSE";
   END_TRANSITION
   STEP Z228_backward:   // S48, max time T#10S, warning time T#7S: Step commentary / Schrittkommentar
      interlock C := "AlwaysFALSE";   // Z228_zur
      supervision V := NOT #Z228__back.TT AND (#Z228_backward.T > T#5S);   // Z228_zur
      (C)     N    "GraDB_SK".noAction
   END_STEP
   TRANSITION Z228__back FROM Z228_backward TO Z229_backward   // T48
      := "AlwaysFALSE";
   END_TRANSITION
   STEP Z229_backward:   // S49, max time T#10S, warning time T#7S: Step commentary / Schrittkommentar
      interlock C := "AlwaysFALSE";   // Z229_zur
      supervision V := NOT #Z229__back.TT AND (#Z229_backward.T > T#5S);   // Z229_zur
      (C)     N    "GraDB_SK".noAction
   END_STEP
   TRANSITION Z229__back FROM Z229_backward TO Z230_backward   // T49
      := "AlwaysFALSE";
   END_TRANSITION
   STEP Z230_backward:   // S50, max time T#10S, warning time T#7S: Step commentary / Schrittkommentar
      interlock C := "AlwaysFALSE";   // Z230_zur
      supervision V := NOT #Z230__back.TT AND (#Z230_backward.T > T#5S);   // Z230_zur
      (C)     N    "GraDB_SK".noAction
   END_STEP
   TRANSITION Z230__back FROM Z230_backward TO Z231_backward   // T50
      := "AlwaysFALSE";
   END_TRANSITION
   STEP Z226_forward:   // S146, max time T#10S, warning time T#7S: Step commentary / Schrittkommentar
      interlock C := "AlwaysFALSE";   // Z226_vor
      supervision V := NOT #Z226_in_front.TT AND (#Z226_forward.T > T#5S);   // Z226_vor
      (C)     N    "GraDB_SK".noAction
   END_STEP
   TRANSITION Z226_in_front FROM Z226_forward TO Z227_forward   // T146
      := "AlwaysFALSE";
   END_TRANSITION
   STEP Z227_forward:   // S147, max time T#10S, warning time T#7S: Step commentary / Schrittkommentar
      interlock C := "AlwaysFALSE";   // Z227_vor
      supervision V := NOT #Z227_in_front.TT AND (#Z227_forward.T > T#5S);   // Z227_vor
      (C)     N    "GraDB_SK".noAction
   END_STEP
   TRANSITION Z227_in_front FROM Z227_forward TO Z228_forward   // T147
      := "AlwaysFALSE";
   END_TRANSITION
   STEP Z228_forward:   // S148, max time T#10S, warning time T#7S: Step commentary / Schrittkommentar
      interlock C := "AlwaysFALSE";   // Z228_vor
      supervision V := NOT #Z228_in_front.TT AND (#Z228_forward.T > T#5S);   // Z228_vor
      (C)     N    "GraDB_SK".noAction
   END_STEP
   TRANSITION Z228_in_front FROM Z228_forward TO Z229_forward   // T148
      := "AlwaysFALSE";
   END_TRANSITION
   STEP Z229_forward:   // S149, max time T#10S, warning time T#7S: Step commentary / Schrittkommentar
      interlock C := "AlwaysFALSE";   // Z229_vor
      supervision V := NOT #Z229_in_front.TT AND (#Z229_forward.T > T#5S);   // Z229_vor
      (C)     N    "GraDB_SK".noAction
   END_STEP
   TRANSITION Z229_in_front FROM Z229_forward TO Z230_forward   // T149
      := "AlwaysFALSE";
   END_TRANSITION
   STEP Z230_forward:   // S150, max time T#10S, warning time T#7S: Step commentary / Schrittkommentar
      interlock C := "AlwaysFALSE";   // Z230_vor
      supervision V := NOT #Z230_in_front.TT AND (#Z230_forward.T > T#5S);   // Z230_vor
      (C)     N    "GraDB_SK".noAction
   END_STEP
   TRANSITION Z230_in_front FROM Z230_forward TO Z231_forward   // T150
      := "AlwaysFALSE";
   END_TRANSITION
   STEP Z231_backward:   // S51, max time T#10S, warning time T#7S: Step commentary / Schrittkommentar
      interlock C := "AlwaysFALSE";   // Z231_zur
      supervision V := NOT #Z231__back.TT AND (#Z231_backward.T > T#5S);   // Z231_zur
      (C)     N    "GraDB_SK".noAction
   END_STEP
   TRANSITION Z231__back FROM Z231_backward TO Z232_backward   // T51
      := "AlwaysFALSE";
   END_TRANSITION
   STEP Z232_backward:   // S52, max time T#10S, warning time T#7S: Step commentary / Schrittkommentar
      interlock C := "AlwaysFALSE";   // Z232_zur
      supervision V := NOT #Z232__back.TT AND (#Z232_backward.T > T#5S);   // Z232_zur
      (C)     N    "GraDB_SK".noAction
   END_STEP
   TRANSITION Z232__back FROM Z232_backward TO Z233_backward   // T52
      := "AlwaysFALSE";
   END_TRANSITION
   STEP Z233_backward:   // S53, max time T#10S, warning time T#7S: Step commentary / Schrittkommentar
      interlock C := "AlwaysFALSE";   // Z233_zur
      supervision V := NOT #Z233__back.TT AND (#Z233_backward.T > T#5S);   // Z233_zur
      (C)     N    "GraDB_SK".noAction
   END_STEP
   TRANSITION Z233__back FROM Z233_backward TO Z234_backward   // T53
      := "AlwaysFALSE";
   END_TRANSITION
   STEP Z234_backward:   // S54, max time T#10S, warning time T#7S: Step commentary / Schrittkommentar
      interlock C := "AlwaysFALSE";   // Z234_zur
      supervision V := NOT #Z234__back.TT AND (#Z234_backward.T > T#5S);   // Z234_zur
      (C)     N    "GraDB_SK".noAction
   END_STEP
   TRANSITION Z234__back FROM Z234_backward TO Z235_backward   // T54
      := "AlwaysFALSE";
   END_TRANSITION
   STEP Z235_backward:   // S55, max time T#10S, warning time T#7S: Step commentary / Schrittkommentar
      interlock C := "AlwaysFALSE";   // Z235_zur
      supervision V := NOT #Z235__back.TT AND (#Z235_backward.T > T#5S);   // Z235_zur
      (C)     N    "GraDB_SK".noAction
   END_STEP
   TRANSITION Z235__back FROM Z235_backward TO Z236_backward   // T55
      := "AlwaysFALSE";
   END_TRANSITION
   STEP Z236_backward:   // S56, max time T#10S, warning time T#7S: Step commentary / Schrittkommentar
      interlock C := "AlwaysFALSE";   // Z236_zur
      supervision V := NOT #Z236__back.TT AND (#Z236_backward.T > T#5S);   // Z236_zur
      (C)     N    "GraDB_SK".noAction
   END_STEP
   TRANSITION Z236__back FROM Z236_backward TO Z237_backward   // T56
      := "AlwaysFALSE";
   END_TRANSITION
   STEP Z237_backward:   // S57, max time T#10S, warning time T#7S: Step commentary / Schrittkommentar
      interlock C := "AlwaysFALSE";   // Z237_zur
      supervision V := NOT #Z237__back.TT AND (#Z237_backward.T > T#5S);   // Z237_zur
      (C)     N    "GraDB_SK".noAction
   END_STEP
   TRANSITION Z237__back FROM Z237_backward TO Z238_backward   // T57
      := "AlwaysFALSE";
   END_TRANSITION
   STEP Z238_backward:   // S58, max time T#10S, warning time T#7S: Step commentary / Schrittkommentar
      interlock C := "AlwaysFALSE";   // Z238_zur
      supervision V := NOT #Z238__back.TT AND (#Z238_backward.T > T#5S);   // Z238_zur
      (C)     N    "GraDB_SK".noAction
   END_STEP
   TRANSITION Z238__back FROM Z238_backward TO Z239_backward   // T58
      := "AlwaysFALSE";
   END_TRANSITION
   STEP Z239_backward:   // S59, max time T#10S, warning time T#7S: Step commentary / Schrittkommentar
      interlock C := "AlwaysFALSE";   // Z239_zur
      supervision V := NOT #Z239__back.TT AND (#Z239_backward.T > T#5S);   // Z239_zur
      (C)     N    "GraDB_SK".noAction
   END_STEP
   TRANSITION Z239__back FROM Z239_backward TO Z240_backward   // T59
      := "AlwaysFALSE";
   END_TRANSITION
   STEP Z240_backward:   // S60, max time T#10S, warning time T#7S: Step commentary / Schrittkommentar
      interlock C := "AlwaysFALSE";   // Z240_zur
      supervision V := NOT #Z240__back.TT AND (#Z240_backward.T > T#5S);   // Z240_zur
      (C)     N    "GraDB_SK".noAction
   END_STEP
   TRANSITION Z240__back FROM Z240_backward TO END   // T60
      := "AlwaysFALSE";
   END_TRANSITION
   STEP Z231_forward:   // S151, max time T#10S, warning time T#7S
      interlock C := "AlwaysFALSE";   // Z231_vor
      supervision V := NOT #Z231_in_front.TT AND (#Z231_forward.T > T#5S);   // Z231_vor
      (C)     N    "GraDB_SK".noAction
   END_STEP
   TRANSITION Z231_in_front FROM Z231_forward TO Z232_forward   // T151
      := "AlwaysFALSE";
   END_TRANSITION
   STEP Z232_forward:   // S152, max time T#10S, warning time T#7S
      interlock C := "AlwaysFALSE";   // Z232_vor
      supervision V := NOT #Z232_in_front.TT AND (#Z232_forward.T > T#5S);   // Z232_vor
      (C)     N    "GraDB_SK".noAction
   END_STEP
   TRANSITION Z232_in_front FROM Z232_forward TO Z233_forward   // T152
      := "AlwaysFALSE";
   END_TRANSITION
   STEP Z233_forward:   // S153, max time T#10S, warning time T#7S
      interlock C := "AlwaysFALSE";   // Z233_vor
      supervision V := NOT #Z233_in_front.TT AND (#Z233_forward.T > T#5S);   // Z233_vor
      (C)     N    "GraDB_SK".noAction
   END_STEP
   TRANSITION Z233_in_front FROM Z233_forward TO Z234_forward   // T153
      := "AlwaysFALSE";
   END_TRANSITION
   STEP Z234_forward:   // S154, max time T#10S, warning time T#7S
      interlock C := "AlwaysFALSE";   // Z234_vor
      supervision V := NOT #Z234_in_front.TT AND (#Z234_forward.T > T#5S);   // Z234_vor
      (C)     N    "GraDB_SK".noAction
   END_STEP
   TRANSITION Z234_in_front FROM Z234_forward TO Z235_forward   // T154
      := "AlwaysFALSE";
   END_TRANSITION
   STEP Z235_forward:   // S155, max time T#10S, warning time T#7S
      interlock C := "AlwaysFALSE";   // Z235_vor
      supervision V := NOT #Z235_in_front.TT AND (#Z235_forward.T > T#5S);   // Z235_vor
      (C)     N    "GraDB_SK".noAction
   END_STEP
   TRANSITION Z235_in_front FROM Z235_forward TO Z236_forward   // T155
      := "AlwaysFALSE";
   END_TRANSITION
   STEP Z236_forward:   // S156, max time T#10S, warning time T#7S: Step commentary / Schrittkommentar
      interlock C := "AlwaysFALSE";   // Z236_vor
      supervision V := NOT #Z236_in_front.TT AND (#Z236_forward.T > T#5S);   // Z236_vor
      (C)     N    "GraDB_SK".noAction
   END_STEP
   TRANSITION Z236_in_front FROM Z236_forward TO Z237_forward   // T156
      := "AlwaysFALSE";
   END_TRANSITION
   STEP Z237_forward:   // S157, max time T#10S, warning time T#7S: Step commentary / Schrittkommentar
      interlock C := "AlwaysFALSE";   // Z237_vor
      supervision V := NOT #Z237_in_front.TT AND (#Z237_forward.T > T#5S);   // Z237_vor
      (C)     N    "GraDB_SK".noAction
   END_STEP
   TRANSITION Z237_in_front FROM Z237_forward TO Z238_forward   // T157
      := "AlwaysFALSE";
   END_TRANSITION
   STEP Z238_forward:   // S158, max time T#10S, warning time T#7S: Step commentary / Schrittkommentar
      interlock C := "AlwaysFALSE";   // Z238_vor
      supervision V := NOT #Z238_in_front.TT AND (#Z238_forward.T > T#5S);   // Z238_vor
      (C)     N    "GraDB_SK".noAction
   END_STEP
   TRANSITION Z238_in_front FROM Z238_forward TO Z239_forward   // T158
      := "AlwaysFALSE";
   END_TRANSITION
   STEP Z239_forward:   // S159, max time T#10S, warning time T#7S: Step commentary / Schrittkommentar
      interlock C := "AlwaysFALSE";   // Z239_vor
      supervision V := NOT #Z239_in_front.TT AND (#Z239_forward.T > T#5S);   // Z239_vor
      (C)     N    "GraDB_SK".noAction
   END_STEP
   TRANSITION Z239_in_front FROM Z239_forward TO Z240_forward   // T159
      := "AlwaysFALSE";
   END_TRANSITION
   STEP Z240_forward:   // S160, max time T#10S, warning time T#7S: Step commentary / Schrittkommentar
      interlock C := "AlwaysFALSE";   // Z240_vor
      supervision V := NOT #Z240_in_front.TT AND (#Z240_forward.T > T#5S);   // Z240_vor
      (C)     N    "GraDB_SK".noAction
   END_STEP
   TRANSITION Z240_in_front FROM Z240_forward TO END   // T160
      := "AlwaysFALSE";
   END_TRANSITION

   // permanent post-instructions
   NETWORK 1
   TITLE = HMI Lite Pass on data / HMI Lite Daten weiterreichen
      "LTLL_ManualGraphInterlock"(ManualGraphExtOutput := #extBlock.output,
                              ManualGraphControlScreen := "LTLL_ManualGraphControl_OP70".screen[0]);
   NETWORK 2
   TITLE = Report step error / Schrittkettenfehler melden
      "SysFC_NumOfSQErrors"(FLT := #RT_DATA.SQ_FLAGS.ERR_FLT,
                            Fault_SQ := "AnwDB_OperatingModes_OP70".BA[0].error_report_SK,
                            NumOf_Fault_SQ := "AnwDB_ZP_Alarm_OP70".FaultsNoSK_ST1);
END_FUNCTION_BLOCK
